// TwinCAT 3 PLC project FMStringsTests
// ProgramVersion: 3.1.4024.0
// libraries:
//   Strings, * (TomasRompotl)
//   Tc2_System, * (Beckhoff Automation GmbH)
//   Tc3_Module, * (Beckhoff Automation GmbH)
//   TcUnit, * (www.tcunit.org)
//   Types, * (TomasRompotl)
// project tree:
//   Builders/ BuildStringInlineTest.TcPOU, StringBuilder255Test.TcPOU, StringBuilderExtBufferTest.TcPOU, StringBuilderInfiniteTest.TcPOU
//   Convert/ ConvertFunctionsTest.TcPOU
//   Manipulate/ ManipulateFunctionsTest.TcPOU
//   / PlcTask.TcTTO (not stored), PRG_Test.TcPOU (not stored)
//   Validate/ ValidateFunctionsTest.TcPOU (not stored)
// (motion and I/O tree: see PLC project fmtypestests)
// real-time tasks:
//   TASK FMTypesTestsTask: cycle T#1ms, priority 20, ADS port 350
//   TASK FMStringsTestsTask: cycle T#1ms, priority 21, ADS port 351
//   TASK FMDataTestsTask: cycle T#1ms, priority 22, ADS port 352
//   TASK FMMathTestsTask: cycle T#1ms, priority 23, ADS port 353
//   TASK FMTimeTestsTask: cycle T#1ms, priority 24, ADS port 354

// ---- Builders/BuildStringInlineTest.TcPOU
FUNCTION_BLOCK BuildStringInlineTest EXTENDS TcUnit.FB_TestSuite
VAR
END_VAR

BuildStringInSingleLine();

METHOD BuildStringInSingleLine : BOOL
VAR
END_VAR
TcUnit.TEST('Build string in single line');

AssertEquals_STRING(
	Expected := '12',
	Actual := BuildStringInline('1').Append('2').GetString(),
	Message := 'Should return built string');

AssertEquals_STRING(
	Expected := 'ab',
	Actual := BuildStringInline('a').Append('b').GetString(),
	Message := 'Should return another built string');

TEST_FINISHED();
END_METHOD

END_FUNCTION_BLOCK

// ---- Builders/StringBuilder255Test.TcPOU
FUNCTION_BLOCK StringBuilder255Test EXTENDS TcUnit.FB_TestSuite
VAR
END_VAR

AppendAndClear();

METHOD AppendAndClear : BOOL
VAR
	builder : StringBuilder255;
END_VAR
TcUnit.TEST('Append and Clear');

builder
	.Clear()
	.Append('1')
	.Append('2');

AssertEquals_STRING(
	Expected := '12',
	Actual := builder.GetString(),
	Message := 'Should return Appended strings using GetString() method');

AssertEquals_STRING(
	Expected := '12',
	Actual := builder.Value,
	Message := 'Should return string using Value property');

AssertEquals_DINT(
	Expected := 2,
	Actual := builder.Length,
	Message := 'Should return string length');	

builder.Clear();

AssertEquals_BOOL(
	Expected := TRUE,
	Actual := builder.IsEmpty,
	Message := 'Should return that string is empty');
	
TEST_FINISHED();
END_METHOD

END_FUNCTION_BLOCK

// ---- Builders/StringBuilderExtBufferTest.TcPOU
FUNCTION_BLOCK StringBuilderExtBufferTest EXTENDS TcUnit.FB_TestSuite
VAR
END_VAR

AppendAndClear();

METHOD AppendAndClear : BOOL
VAR
	buffer : STRING(2000);
	builder : StringBuilderExtBuffer := (Buffer := ToAnyType(buffer));
	
	testValue : STRING := ' very long strings';
END_VAR
TcUnit.TEST('Append and Clear');

builder
	.Clear()
	.Append('SB with external buffer')
	.Append(' is meant for')
	.AppendByPointer(ADR(testValue));

AssertEquals_STRING(
	Expected := 'SB with external buffer is meant for very long strings',
	Actual := buffer,
	Message := 'Strings should be properly appended');

builder.Clear();

AssertEquals_BOOL(
	Expected := TRUE,
	Actual := builder.IsEmpty,
	Message := 'Buffer should be empty');
	
TEST_FINISHED();
END_METHOD

END_FUNCTION_BLOCK

// ---- Builders/StringBuilderInfiniteTest.TcPOU
FUNCTION_BLOCK StringBuilderInfiniteTest EXTENDS TcUnit.FB_TestSuite
VAR
END_VAR

AppendAndClear();
CheckCapacityHasIncreased();

METHOD AppendAndClear : BOOL
VAR
	builder : StringBuilderInfinite;
	testValue : STRING := ' very long strings without care';
END_VAR
TcUnit.TEST('Append and Clear');

builder
	.Clear()
	.Append('SB infinite')
	.Append(' is meant for')
	.AppendByPointer(ADR(testValue));

AssertEquals_STRING(
	Expected := 'SB infinite is meant for very long strings without care',
	Actual := builder.Value^,
	Message := 'Strings should be properly appended');

builder.Clear();

AssertEquals_BOOL(
	Expected := TRUE,
	Actual := builder.IsEmpty,
	Message := 'String should be empty');
	
TEST_FINISHED();
END_METHOD

METHOD CheckCapacityHasIncreased : BOOL
VAR
	builder : StringBuilderInfinite;
	i : INT;
END_VAR
TcUnit.TEST('Check capacity has increased');

AssertEquals_DINT(
	Expected := 1024,
	Actual := builder.Capacity,
	Message := 'Initial capacity should be 1000');
	
builder.Clear();
FOR i := 0 TO 999 DO
	builder.Append('0123456789');
END_FOR

AssertEquals_DINT(
	Expected := 10000,
	Actual := builder.Length,
	Message := 'String should be 10000 long');

AssertEquals_DINT(
	Expected := 16384,
	Actual := builder.Capacity,
	Message := 'Capacity should be increased to 16384');
	
TEST_FINISHED();
END_METHOD

END_FUNCTION_BLOCK

// ---- Convert/ConvertFunctionsTest.TcPOU
FUNCTION_BLOCK ConvertFunctionsTest EXTENDS TcUnit.FB_TestSuite
VAR
END_VAR

AnyTypeToStringFunction();
StringToAnyFunction();

METHOD AnyTypeToStringFunction : BOOL
VAR
	stringVar : T_MaxString := 'test';
	intVar : INT := 42;
	realVar : REAL := 3.14;
END_VAR
TcUnit.TEST('ANY to STRING');

AssertEquals_STRING(
	Expected := 'test',
	Actual := AnyToString(stringVar),
	Message := 'Should convert STRING var to STRING');

AssertEquals_STRING(
	Expected := '42',
	Actual := AnyToString(intVar),
	Message := 'Should convert INT var to STRING');

AssertEquals_STRING(
	Expected := '3.14',
	Actual := AnyToString(realVar),
	Message := 'Should convert REAL var to STRING');
	
TEST_FINISHED();
END_METHOD

METHOD StringToAnyFunction : BOOL
VAR
	stringVar : T_MaxString;
	intVar : INT;
	realVar : REAL;
END_VAR
TcUnit.TEST('STRING to ANY');

StringToAny('this is test', stringVar);
StringToAny('42', intVar);
StringToAny('3.14', realVar);

AssertEquals_STRING(
	Expected := 'this is test',
	Actual := stringVar,
	Message := 'Should return correct STRING value');

AssertEquals_INT(
	Expected := 42,
	Actual := intVar,
	Message := 'Should return correct INT value');

AssertEquals_REAL(
	Expected := 3.14,
	Actual := realVar,
	Delta := 0.001,
	Message := 'Should return correct REAL value');

TEST_FINISHED();
END_METHOD

END_FUNCTION_BLOCK

// ---- Manipulate/ManipulateFunctionsTest.TcPOU
FUNCTION_BLOCK ManipulateFunctionsTest EXTENDS TcUnit.FB_TestSuite
VAR
END_VAR

AddLeadingZerosFunction();
GetStringBetweenFunction();
RemoveStringFromEndFunction();
ReplaceStringFunction();

METHOD AddLeadingZerosFunction : BOOL
VAR
	test : T_MaxString := '555';
END_VAR
TcUnit.TEST('Add leading zeros');

AssertEquals_STRING(
	Expected := '00555',
	Actual := AddLeadingZeros(test, 5),
	Message := 'Should pad propper number of zeros');

AssertEquals_STRING(
	Expected := '555',
	Actual := AddLeadingZeros(test, 2),
	Message := 'Should do nothing if formatter string already has more chars');

TEST_FINISHED();
END_METHOD

METHOD GetStringBetweenFunction : BOOL
VAR
	test0 : T_MaxString := '1';
	test1 : T_MaxString := '[2]';
	test2 : T_MaxString := 'TestValue[3]rest';
	actual : T_MaxString;
END_VAR
TcUnit.TEST('Get string between');

actual := GetStringBetween(test0, '[', ']');

AssertEquals_STRING(
	Expected := '',
	Actual := actual,
	Message := 'Should return nothing');

actual := GetStringBetween(test1, '[', ']');

AssertEquals_STRING(
	Expected := '2',
	Actual := actual,
	Message := 'Should return content of brackets');

actual := GetStringBetween(test2, '[', ']');

AssertEquals_STRING(
	Expected := '3',
	Actual := actual,
	Message := 'Should return content of brackets');

TEST_FINISHED();
END_METHOD

METHOD RemoveStringFromEndFunction : BOOL
VAR
	test : T_MaxString := 'Last word will be removed';
	actual : T_MaxString;
END_VAR
TcUnit.TEST('Remove string from end');

actual := RemoveStringFromEnd(test, 'removed');

AssertEquals_STRING(
	Expected := 'Last word will be ',
	Actual := actual,
	Message := 'Should remove last word from test string');

TEST_FINISHED();
END_METHOD

METHOD ReplaceStringFunction : BOOL
VAR
	test : T_MaxString := 'this is test string';
END_VAR
TcUnit.TEST('Replace string');

ReplaceString(test, 'not here', 'replaced');

AssertEquals_STRING(
	Expected := 'this is test string',
	Actual := test,
	Message := 'Should do nothing because searched string is not there');

ReplaceString(test, 'test', 'replaced');

AssertEquals_STRING(
	Expected := 'this is replaced string',
	Actual := test,
	Message := 'Should replace found string');

TEST_FINISHED();
END_METHOD

END_FUNCTION_BLOCK
